FUNCTION_BLOCK _TemplateTest EXTENDS TcUnit.FB_TestSuite
VAR
END_VAR

ExampleTest();

METHOD ExampleTest : BOOL
VAR
	expected : INT;
	actual : INT;
END_VAR
TcUnit.TEST('Example test');

expected := ;
actual := ;

AssertEquals(
	Expected := expected,
	Actual := actual,
	Message := 'What went wrong');

TEST_FINISHED();
END_METHOD

END_FUNCTION_BLOCK

(* stored: Version 1.1.0.1, ProductVersion 3.1.4024.12
   POU _TemplateTest: Id {e4bd020e-6073-0bd1-2b98-9e2be6ba5528}, SpecialFunc None
   Method ExampleTest: Id {3cde1621-eda1-0408-1ed2-428c81e7feb8} *)
